{attribute 'qualified_only'}
VAR_GLOBAL
	value1:DINT;
END_VAR

(* stored: Version 1.1.0.1, ProductVersion 3.1.4023.14
   GVL GVL1: Id {79bdcdcb-4dc2-471e-a816-01594a962c56} *)
